TYPE aT_Heater :
STRUCT
	InPressure: REAL;
	InFlow: REAL;
	Temperature: REAL;
	Pressure: REAL;
END_STRUCT
END_TYPE

(* stored: Version 1.1.0.1, ProductVersion 3.1.4024.4
   DUT aT_Heater: Id {e265f4f9-b794-4e10-8e46-4998168107cb} *)
